# EPICS IOC start-up script: iocsh/ethercatmcTestInputRecordAlarm.iocsh
ethercatmcCreateAsynParam $(MOTOR_PORT) DISCRETEINPUT Int32
ethercatmcCreateAsynParam $(MOTOR_PORT) DISCRETEINPUT_StatusBits UInt32Digital
ethercatmcCreateAsynParam $(MOTOR_PORT) DISCRETEOUTPUT Int32

dbLoadRecords("ethercatmcTestInputRecordAlarm.template", "SYSPFX=$(SYSPFX), AXIS_NAME=$(AXIS_NAME), MOTOR_PORT=$(MOTOR_PORT), AXIS_NO=$(AXIS_NO)")
